(* CoDeSys 2.3.9.26 project: Assignment.pro *)
(* Libraries: Standard.LIB 4.10.05 11:14:46, Util.lib 18.5.10 15:14:28 *)

(* POU PLC_PRG, ST *)
PROGRAM PLC_PRG
VAR
	TimeOfDay:TOD;

	(*Input*)
	Start: BOOL;
	LS2: BOOL;
	LS1: BOOL;
	heater_start: BOOL;
	in_flow_value:REAL;
	Heater:BOOL;
	input_slider:REAL;
	input_slider2:DINT;
	drain_slider:REAL;
	drain_slider2:DINT;
	TankTemp_slider:REAL;
	TankTemp_slider2:DINT;
	Tank_Temp:DINT;

	(*Output*)
	heat_ton1: TON;
	out_valve: BOOL;
	in_valve: BOOL;

	(*Water Height Calculation*)
	tank_fill: REAL;
	FreshWaterTemp:REAL;
	TankArea: REAL;
	Pi: REAL;
	Radius: REAL;
	WaterHeight: REAL;
	WaterHeight2:DINT;

	(*Water in tank Final Temp calculation*)
	HeatedWaterV1:REAL;
	HeatedWaterT1:REAL;
	ChilledWaterV2:REAL;
	ChilledWaterT2:REAL;
	Water_Tfinal:REAL;

	(*Heater*)
	TimeToHeat: REAL;
	CurrentWaterVolume: REAL; (*In Litres*)
	TargetTempFreshTempDifference: REAL;
	Numerator: REAL;
	Numerator2: REAL;
	heat_timer: BOOL;
END_VAR
(*---Water Height Calculation-----*)
(*1drum/200litres = 58cm*90cm*)
(*Let's say 200 litres tank, therefore 200000 millilitres*)
(*Flow rate = 1 litre per minute if value is set to 1*)
(*TankVolume=pi*radius*radius*height*)
Pi:=3.14;
Radius:=29; (*In centimeters*)
TankArea:=Pi*(Radius*Radius);
WaterHeight:=(tank_fill/TankArea); (*tank_fill is in cubic cm*)
WaterHeight2:=REAL_TO_DINT(WaterHeight);
(*--------------------------------*)



(*-----------Initialize-----------*)
IF Start=FALSE THEN
	in_valve:=FALSE;
	LS1:=FALSE;
	LS2:=FALSE;
	heater_start:=FALSE;
	out_valve:=FALSE;
END_IF
(*--------------------------------*)


(*---------Filling Control--------*)
input_slider2:=REAL_TO_DINT(input_slider);

IF in_valve=TRUE THEN
	tank_fill:=tank_fill+input_slider;
ELSE
	tank_fill:=tank_fill+0;
END_IF

IF tank_fill>=200000 THEN
	LS2:=TRUE;
	in_valve:=FALSE;
ELSE
	LS2:=FALSE;
END_IF
(*--------------------------------*)


(*--------Emptying Control--------*)
drain_slider2:=REAL_TO_DINT(drain_slider);

IF out_valve=TRUE THEN
	tank_fill:=tank_fill-drain_slider;
ELSE
	tank_fill:=tank_fill-0;
END_IF

IF tank_fill<=0 THEN
	LS1:=FALSE;
	out_valve:=FALSE;
	(*in_valve:=TRUE;*)
	heater_start:=FALSE;
ELSE
	LS1:=TRUE;
END_IF
(*--------------------------------*)

(*-----Heating Control------------*)
TankTemp_slider2:=REAL_TO_DINT(TankTemp_slider);

IF heater_start=1 THEN
	Tank_Temp:=TankTemp_slider2;
ELSE
	Tank_Temp:=Tank_Temp-1;
END_IF

IF Tank_Temp<24 THEN
	Tank_Temp:=24;
END_IF

IF heater_start=1 THEN
	heat_ton1(IN:=TRUE, PT:=t#10000s);
	heat_timer:=heat_ton1.Q;
END_IF

IF TankTemp_slider>=100 THEN
	heater_start:=FALSE;
END_IF

(*--------------------------------*)


(*----Time to Heat Calculation-----
FreshWaterTemp:=24;(*In degree Celsius*)
(*TimeToHeat(hours):=((4.2*WaterVolume*(TargetTemp-FreshWaterTemp))/3600)*HeaterWattage(kW)*)
CurrentWaterVolume:=tank_fill/1000; (*Value in litres*)
TargetTempFreshTempDifference:=100-FreshWaterTemp;
Numerator:=4.2*CurrentWaterVolume*TargetTempFreshTempDifference;
Numerator2:=Numerator/3600;
TimeToHeat:=Numerator2/100;
TimeOfDay:=tod#00:00:00;
--------------------------------*)


(*---Tank Temp Calculation----*)
(*HeatCap:=(ThermalEnergyinJoules)/(MassInKG*TempInCelsius)*)
(*Tfinal=((V1*Thot)+(V2*Tcold))/(V1+V2)*)
(*Water_Tfinal:=((HeatedWaterV1*HeatedWaterT1)+(ChilledWaterV2*ChilledWaterT2))/(HeatedWaterV1+ChilledWaterV2);*)
(*--------------------------------*)
END_PROGRAM

(* Visualisation HMI
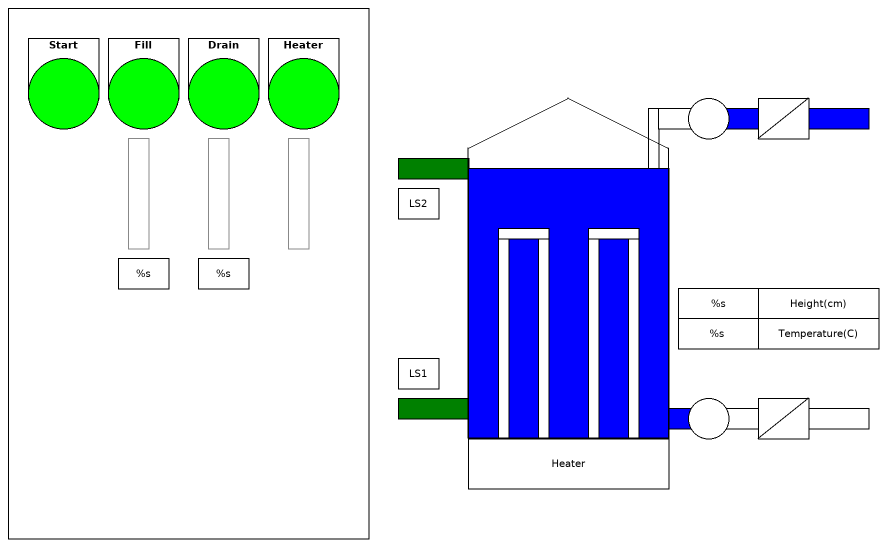
rectangle at (650,110)-(661,431): invisible if PLC_PRG.in_valve=FALSE; alarm colour if PLC_PRG.in_valve; toggles PLC_PRG.in_valve
rectangle at (30,40)-(101,101): text "Start"
rectangle at (720,410)-(871,431): alarm colour if PLC_PRG.out_valve
ellipse at (30,60)-(101,131): alarm colour if PLC_PRG.Start; toggles PLC_PRG.Start
rectangle at (660,110)-(701,131): alarm colour if PLC_PRG.in_valve; toggles PLC_PRG.in_valve
ellipse at (690,100)-(731,141): alarm colour if PLC_PRG.in_valve
other8 at (130,140)-(151,251): dynamic style PLC_PRG.in_flow_value
rectangle at (470,440)-(671,491): text "Heater"; alarm colour if PLC_PRG.heater_start
ellipse at (690,400)-(731,441): alarm colour if PLC_PRG.out_valve
rectangle at (400,190)-(441,221): text "LS2"; alarm colour if PLC_PRG.LS2; toggles PLC_PRG.LS2
rectangle at (400,360)-(441,391): text "LS1"; alarm colour if PLC_PRG.LS1; toggles PLC_PRG.LS1
rectangle at (470,420)-(671,441): invisible if PLC_PRG.tank_fill<0
rectangle at (470,360)-(671,441): invisible if PLC_PRG.tank_fill<50000
rectangle at (470,290)-(671,441): invisible if PLC_PRG.tank_fill<100000
rectangle at (470,230)-(671,441): invisible if PLC_PRG.tank_fill<150000
rectangle at (470,170)-(671,441): invisible if PLC_PRG.tank_fill<200000
rectangle at (680,290)-(761,321): text "%s"; shows PLC_PRG.WaterHeight2
rectangle at (680,320)-(761,351): text "%s"; shows PLC_PRG.Tank_Temp
rectangle at (760,290)-(881,321): text "Height(cm)"
rectangle at (760,320)-(881,351): text "Temperature(C)"
rectangle at (500,240)-(511,441): alarm colour if PLC_PRG.heater_start
rectangle at (540,240)-(551,441): alarm colour if PLC_PRG.heater_start
rectangle at (590,240)-(601,441): alarm colour if PLC_PRG.heater_start
rectangle at (500,230)-(551,241): alarm colour if PLC_PRG.heater_start
rectangle at (630,240)-(641,441): alarm colour if PLC_PRG.heater_start
rectangle at (590,230)-(641,241): alarm colour if PLC_PRG.heater_start
rectangle at (270,40)-(341,101): text "Heater"
ellipse at (270,60)-(341,131): alarm colour if PLC_PRG.heater_start; toggles PLC_PRG.heater_start
rectangle at (110,40)-(181,101): text "Fill"
ellipse at (110,60)-(181,131): alarm colour if PLC_PRG.in_valve; toggles PLC_PRG.in_valve
rectangle at (190,40)-(261,101): text "Drain"
ellipse at (190,60)-(261,131): alarm colour if PLC_PRG.out_valve; toggles PLC_PRG.out_valve
rectangle at (120,260)-(171,291): text "%s"; shows PLC_PRG.input_slider2
rectangle at (200,260)-(251,291): text "%s"; shows PLC_PRG.drain_slider2
13 more shapes without text or variables
1 elements of other kinds (tables, trends, ...) not read
*)
